INTERFACE IPointerEnumerable EXTENDS IObject

METHOD GetDefaultEnumerator : IPointerEnumerator
END_METHOD

END_INTERFACE

(* stored: Version 1.1.0.1
   Itf IPointerEnumerable: Id {e960eecd-5ff1-4da6-881f-fa217c428eab}
   Method GetDefaultEnumerator: Id {60ca34a9-85ab-4cf1-83bb-0895f131ec56} *)
